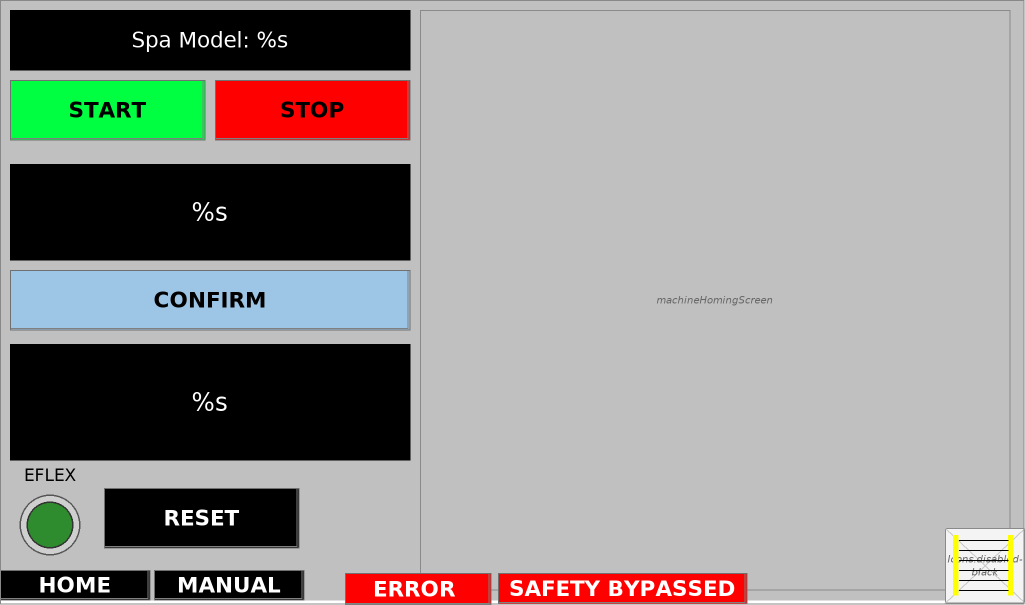
VISUALIZATION eflexScreen  // 1025x605
    Rectangle (0,0 1024x600)
    Button (0,570 150x30), "HOME"
        OnMouseDown: change screen: mainScreen
        OnMouseDown: execute { GVL_machine.nPageIndex := 0; }
    Button (154,570 150x30), "MANUAL"
        OnMouseDown: change screen: manualScreen
        OnMouseDown: execute { GVL_machine.nPageIndex := 5; }
    RoundedRectangle (10,10 400x60), "Spa Model: %s", text variable: GVL_eflex.sSpaModel
    Button (10,80 195x60), "START", invisible if: auto.bHideStartBtn
        toggle auto.bStartBtn
    Button (215,80 195x60), "STOP", invisible if: auto.bHideStopBtn
        toggle auto.bStopBtn
    Frame (420,10 590x580), frame switch variable: auto.nFrameDisp
        shows machineHomingScreen()
        shows baseInSkiOutScreen()
        shows loadSpaScreen()
        shows studsInScreen()
        shows unloadSpaScreen()
        shows manualScreen()
        shows safetyResetScreen()
        shows tempEflexScreen()
        shows continueAutoScreen()
    Textfield (10,164 400x96), "%s", text variable: auto.sPromptDisp
    Button (10,270 400x60), "CONFIRM", invisible if: auto.bHideConfirmBtn
        tap auto.bConfirmBtn
    RoundedRectangle (0,460 100x30), "EFLEX"
    Lamp1 (15,490 70x70), variable: eflex.fbMqttClient.bConnected, style: Lamp-Lamp1-Green
    Button (104,488 195x60), "RESET"
        toggle auto.bResetBtn
    Button (498,573 249x31), "SAFETY BYPASSED", invisible if: NOT GVL_machine.bSafetyBypass
        OnMouseDown: change screen: safetyDisableWarning
    Button (345,573 146x32), "ERROR", invisible if: NOT GVL_machine.bDispErrorIcon
        OnMouseDown: change screen: errorScreen
    Image (945,528 80x75), invisible if: MAIN.bHideLtCurtainDisable, image: Icons.disabled-black
    Group (953,535 60x60), invisible if: GVL_machine.bSafetyBypass
        toggle GVL_machine.bMuteSafety
        Rectangle (0,0 5x60)
        Rectangle (55,0 5x60)
        Line (6,5) (55,5)
        Line (6,15) (55,15)
        Line (6,25) (55,25)
        Line (6,35) (55,35)
        Line (6,45) (55,45)
        Line (6,55) (55,55)
    Textfield (10,344 400x116), "%s", text variable: auto.sCheckDisp, invisible if: auto.bHideCheckDisp
END_VISUALIZATION

(* stored: Version 1.1.0.1, ProductVersion 3.1.4024.13
   Visu eflexScreen: Id {9761f504-d517-4457-b961-c4b8cc78316e} *)
